FUNCTION F_MeterToSubPixelReal : LREAL
VAR_INPUT
  fPosMeter   : LREAL;             (*Position or distance in [m]*)
  fResoSubPx  : LREAL;             (*SubPixel resolution [dpi*SubPx]*)
END_VAR

F_MeterToSubPixelReal := (((fPosMeter * fResoSubPx) / 0.0254));

END_FUNCTION

(* stored: Version 1.1.0.1, ProductVersion 3.1.4024.3
   POU F_MeterToSubPixelReal: Id {ff12f9cd-2d36-4cd6-b1f4-11ff551a2c2d}, SpecialFunc None *)
